// TwinCAT 3 PLC project Untitled1
// ProgramVersion: 3.1.4023.0
// libraries:
//   Pushover, * (Stefan Besler)
//   Tc2_Standard, * (Beckhoff Automation GmbH)
//   Tc2_System, * (Beckhoff Automation GmbH)
//   Tc3_Module, * (Beckhoff Automation GmbH)
// project tree:
//   / PlcTask.TcTTO
//   POUs/ MAIN.TcPOU
// real-time tasks:
//   TASK PlcTask: cycle T#10ms, priority 20, ADS port 350

CONFIGURATION Untitled1
    RESOURCE PLC ON TwinCAT3
        TASK PlcTask(INTERVAL := T#10ms, PRIORITY := 20);
        PROGRAM MAIN WITH PlcTask : MAIN;
    END_RESOURCE
END_CONFIGURATION

// ---- POUs/MAIN.TcPOU
PROGRAM MAIN
VAR
  _step : INT;
  _pushoverClient : Pushover.PushoverClient('<your_api_token>', '<your_user_token>'); 
  _send : BOOL;
END_VAR



IF _send
THEN
  _send := FALSE;
  _step := 10;
END_IF

CASE _step
OF
  0:
    //_pushover.Host := '192.168.1.100'; // specify host if local Pushover ADS Server is running on a different host
    //_pushover.Port := 80080; // specify port if local Pushover ADS Server is running on a non-default port
    
  10:
    _pushoverClient.SendMessageAsync('PLC1', 'Hello World!');
    _step := 20;
    
  20:
    _pushoverClient.Cyclic();
  
    IF _pushoverClient.Error
    THEN
      _step := 99;
    ELSIF NOT _pushoverClient.Busy
    THEN
      _step := 20;
		END_IF
    
  30: // Success
    ;
    
  99: // Error
    ;
END_CASE

END_PROGRAM
